// TIA Portal V17 export
// export: Created 2024-09-27T18:53:45.8218264Z, ExportSetting WithDefaults, DisplayName Totally Integrated Automation Portal, DisplayVersion V17, DisplayName TIA Portal Openness, DisplayVersion V17, DisplayName TIA Portal Version Control Interface, DisplayVersion V17, DisplayName STEP 7 Professional, DisplayVersion V17, DisplayName STEP 7 Safety, DisplayVersion V17, DisplayName WinCC Professional, DisplayVersion V17
FUNCTION "USTAWIENIA" : Void   // FC3, LAD
{ S7_Optimized_Access := 'TRUE' }
VERSION : 0.1
// stored: AutoNumber true, IsIECCheckEnabled false, SetENOAutomatically false, UDAEnableTagReadback false
   VAR_TEMP
      temp_calc_new_tact2 : DInt;
      temp_calc_3 : DInt;
      temp_calc4 : Real;
      temp_calc5 : DInt;
      temp_calc6 : DInt;
      m_zboczeP_ustaw_czas_ssania : Bool;
      temp_calc7 : Real;
      temp_calc8 : Real;
      temp_calc9 : Real;
      temp_calc10 : DInt;
      temp_calc11 : DInt;
      temp_calc12 : Real;
      temp_calc13 : Real;
      temp_calc14 : DInt;
      temp_calc15 : DInt;
      temp_calc16 : Real;
      temp_calc17 : Real;
      temp_calc18 : DInt;
      temp_calc19 : DInt;
      temp_calc20 : Real;
      m_zboczeN_ustaw_delay_zag : Bool;
      m_zboczeN_ustaw_delay_odb : Bool;
      m_zbocze_P_ustaw_delay_odbior : Bool;
   END_VAR
   VAR_TEMP   // added for the SCL form of the ladder/FBD networks
      _w1 : Bool;
      _w2 : Bool;
      _w3 : Bool;
      _w4 : Bool;
      _w5 : Bool;
      _w6 : Bool;
   END_VAR
BEGIN

REGION Network 1: KASOWANIE LICZNIKÓW ZADANYCH SZTUK I WYKONANYCH
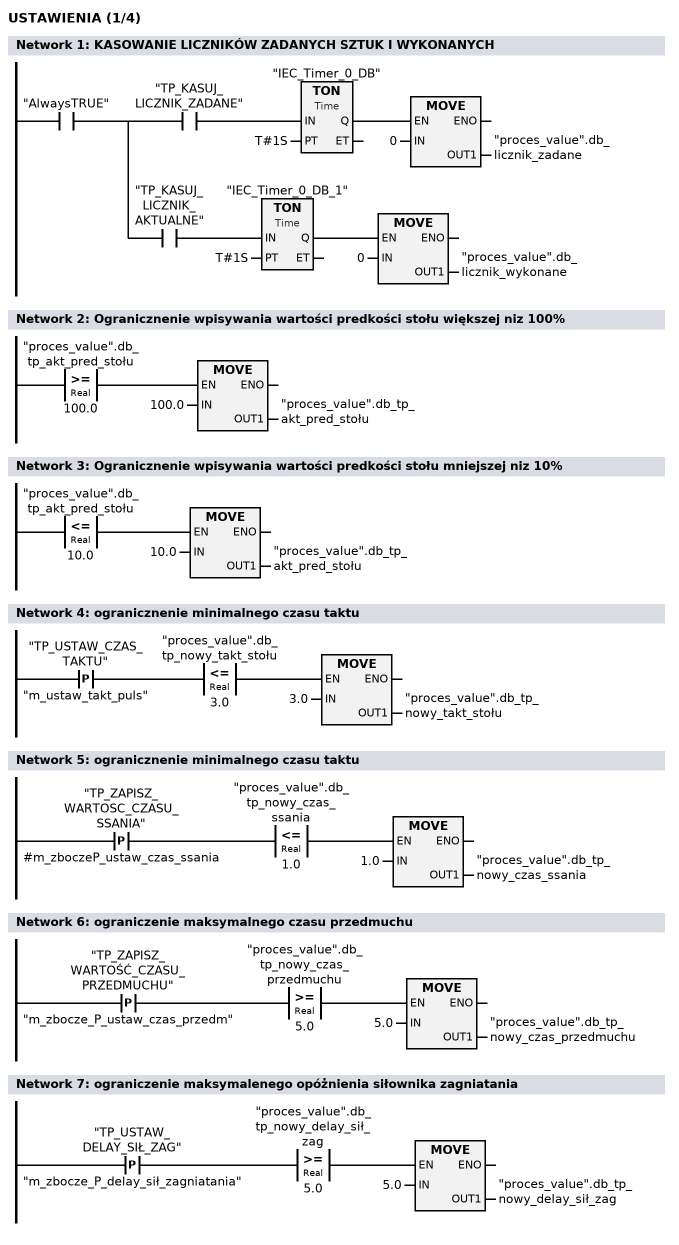
   RUNG wire#powerrail
      Contact( "AlwaysTRUE" )
      wire#w1
      Contact( "TP_KASUJ_LICZNIK_ZADANE" )
      { S7_Templates := "time_type := Time" } "IEC_Timer_0_DB".TON(pt := T#1S, et =>)
      Move(in := 0, out1 => "proces_value".db_licznik_zadane)
   END_RUNG
   RUNG wire#w1
      Contact( "TP_KASUJ_LICZNIK_AKTUALNE" )
      { S7_Templates := "time_type := Time" } "IEC_Timer_0_DB_1".TON(pt := T#1S, et =>)
      Move(in := 0, out1 => "proces_value".db_licznik_wykonane)
   END_RUNG
   // the same network as SCL:
   "IEC_Timer_0_DB".TON(IN := "AlwaysTRUE" AND "TP_KASUJ_LICZNIK_ZADANE", PT := T#1S);
   IF "IEC_Timer_0_DB".Q THEN "proces_value".db_licznik_zadane := 0; END_IF;
   "IEC_Timer_0_DB_1".TON(IN := "AlwaysTRUE" AND "TP_KASUJ_LICZNIK_AKTUALNE", PT := T#1S);
   IF "IEC_Timer_0_DB_1".Q THEN "proces_value".db_licznik_wykonane := 0; END_IF;
END_REGION

REGION Network 2: Ogranicznenie wpisywania wartości predkości stołu większej niz 100%
   RUNG wire#powerrail
      { S7_Templates := "SrcType := Real" } GE_Contact(in1 := "proces_value".db_tp_akt_pred_stołu, in2 := 100.0)
      Move(in := 100.0, out1 => "proces_value".db_tp_akt_pred_stołu)
   END_RUNG
   // the same network as SCL:
   IF "proces_value".db_tp_akt_pred_stołu >= 100.0 THEN "proces_value".db_tp_akt_pred_stołu := 100.0; END_IF;
END_REGION

REGION Network 3: Ogranicznenie wpisywania wartości predkości stołu mniejszej niz 10%
   RUNG wire#powerrail
      { S7_Templates := "SrcType := Real" } LE_Contact(in1 := "proces_value".db_tp_akt_pred_stołu, in2 := 10.0)
      Move(in := 10.0, out1 => "proces_value".db_tp_akt_pred_stołu)
   END_RUNG
   // the same network as SCL:
   IF "proces_value".db_tp_akt_pred_stołu <= 10.0 THEN "proces_value".db_tp_akt_pred_stołu := 10.0; END_IF;
END_REGION

REGION Network 4: ogranicznenie minimalnego czasu taktu
   RUNG wire#powerrail
      P_Contact(operand := "TP_USTAW_CZAS_TAKTU", bit := "m_ustaw_takt_puls")
      { S7_Templates := "SrcType := Real" } LE_Contact(in1 := "proces_value".db_tp_nowy_takt_stołu, in2 := 3.0)
      Move(in := 3.0, out1 => "proces_value".db_tp_nowy_takt_stołu)
   END_RUNG
   // the same network as SCL:
   #_w1 := "TP_USTAW_CZAS_TAKTU" AND NOT "m_ustaw_takt_puls";   // rising edge of "TP_USTAW_CZAS_TAKTU"
   "m_ustaw_takt_puls" := "TP_USTAW_CZAS_TAKTU";
   IF #_w1 AND ("proces_value".db_tp_nowy_takt_stołu <= 3.0) THEN
       "proces_value".db_tp_nowy_takt_stołu := 3.0;
   END_IF;
END_REGION

REGION Network 5: ogranicznenie minimalnego czasu taktu
   RUNG wire#powerrail
      P_Contact(operand := "TP_ZAPISZ_WARTOSC_CZASU_SSANIA", bit := #m_zboczeP_ustaw_czas_ssania)
      { S7_Templates := "SrcType := Real" } LE_Contact(in1 := "proces_value".db_tp_nowy_czas_ssania, in2 := 1.0)
      Move(in := 1.0, out1 => "proces_value".db_tp_nowy_czas_ssania)
   END_RUNG
   // the same network as SCL:
   #_w1 := "TP_ZAPISZ_WARTOSC_CZASU_SSANIA" AND NOT #m_zboczeP_ustaw_czas_ssania;   // rising edge of "TP_ZAPISZ_WARTOSC_CZASU_SSANIA"
   #m_zboczeP_ustaw_czas_ssania := "TP_ZAPISZ_WARTOSC_CZASU_SSANIA";
   IF #_w1 AND ("proces_value".db_tp_nowy_czas_ssania <= 1.0) THEN
       "proces_value".db_tp_nowy_czas_ssania := 1.0;
   END_IF;
END_REGION

REGION Network 6: ograniczenie maksymalnego czasu przedmuchu
   RUNG wire#powerrail
      P_Contact(operand := "TP_ZAPISZ_WARTOŚĆ_CZASU_PRZEDMUCHU", bit := "m_zbocze_P_ustaw_czas_przedm")
      { S7_Templates := "SrcType := Real" } GE_Contact(in1 := "proces_value".db_tp_nowy_czas_przedmuchu, in2 := 5.0)
      Move(in := 5.0, out1 => "proces_value".db_tp_nowy_czas_przedmuchu)
   END_RUNG
   // the same network as SCL:
   #_w1 := "TP_ZAPISZ_WARTOŚĆ_CZASU_PRZEDMUCHU" AND NOT "m_zbocze_P_ustaw_czas_przedm";   // rising edge of "TP_ZAPISZ_WARTOŚĆ_CZASU_PRZEDMUCHU"
   "m_zbocze_P_ustaw_czas_przedm" := "TP_ZAPISZ_WARTOŚĆ_CZASU_PRZEDMUCHU";
   IF #_w1 AND ("proces_value".db_tp_nowy_czas_przedmuchu >= 5.0) THEN
       "proces_value".db_tp_nowy_czas_przedmuchu := 5.0;
   END_IF;
END_REGION

REGION Network 7: ograniczenie maksymalenego opóżnienia siłownika zagniatania
   RUNG wire#powerrail
      P_Contact(operand := "TP_USTAW_DELAY_SIŁ_ZAG", bit := "m_zbocze_P_delay_sił_zagniatania")
      { S7_Templates := "SrcType := Real" } GE_Contact(in1 := "proces_value".db_tp_nowy_delay_sił_zag, in2 := 5.0)
      Move(in := 5.0, out1 => "proces_value".db_tp_nowy_delay_sił_zag)
   END_RUNG
   // the same network as SCL:
   #_w1 := "TP_USTAW_DELAY_SIŁ_ZAG" AND NOT "m_zbocze_P_delay_sił_zagniatania";   // rising edge of "TP_USTAW_DELAY_SIŁ_ZAG"
   "m_zbocze_P_delay_sił_zagniatania" := "TP_USTAW_DELAY_SIŁ_ZAG";
   IF #_w1 AND ("proces_value".db_tp_nowy_delay_sił_zag >= 5.0) THEN
       "proces_value".db_tp_nowy_delay_sił_zag := 5.0;
   END_IF;
END_REGION

REGION Network 8: ograniczenie maksymalenego opóżnienia siłownika odbioru
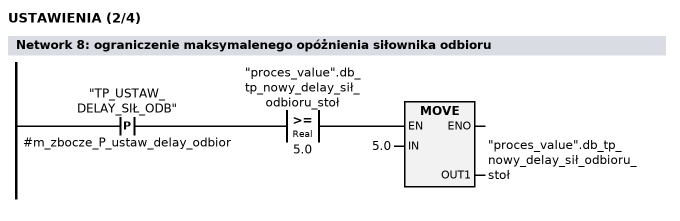
   RUNG wire#powerrail
      P_Contact(operand := "TP_USTAW_DELAY_SIŁ_ODB", bit := #m_zbocze_P_ustaw_delay_odbior)
      { S7_Templates := "SrcType := Real" } GE_Contact(in1 := "proces_value".db_tp_nowy_delay_sił_odbioru_stoł, in2 := 5.0)
      Move(in := 5.0, out1 => "proces_value".db_tp_nowy_delay_sił_odbioru_stoł)
   END_RUNG
   // the same network as SCL:
   #_w1 := "TP_USTAW_DELAY_SIŁ_ODB" AND NOT #m_zbocze_P_ustaw_delay_odbior;   // rising edge of "TP_USTAW_DELAY_SIŁ_ODB"
   #m_zbocze_P_ustaw_delay_odbior := "TP_USTAW_DELAY_SIŁ_ODB";
   IF #_w1 AND ("proces_value".db_tp_nowy_delay_sił_odbioru_stoł >= 5.0) THEN
       "proces_value".db_tp_nowy_delay_sił_odbioru_stoł := 5.0;
   END_IF;
END_REGION

REGION Network 9: OBSŁUGA LICZNIKÓW I TIMERÓW
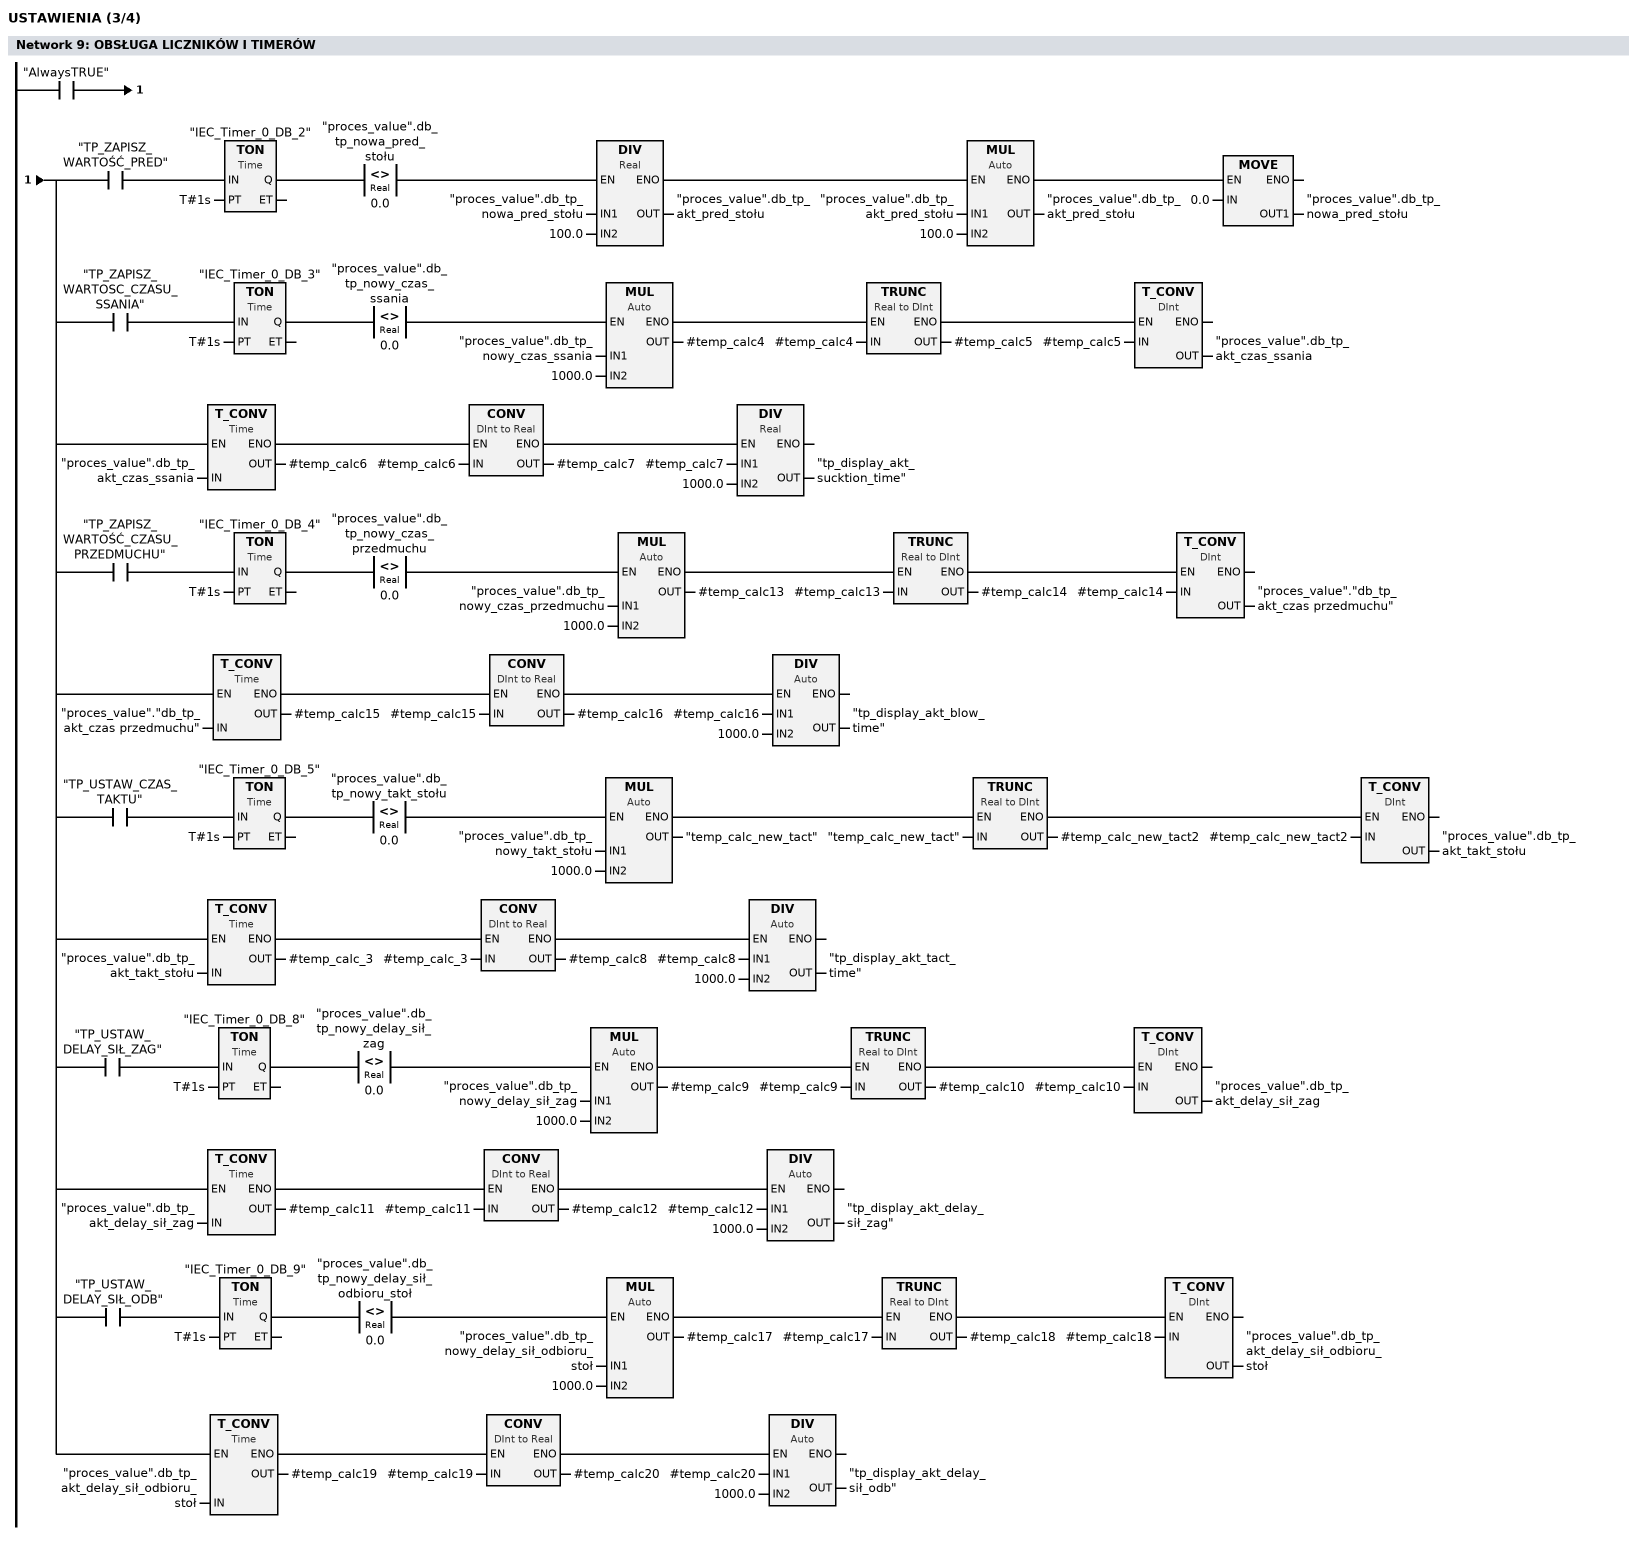
   RUNG wire#powerrail
      Contact( "AlwaysTRUE" )
      wire#w1
      Contact( "TP_ZAPISZ_WARTOŚĆ_PRED" )
      { S7_Templates := "time_type := Time" } "IEC_Timer_0_DB_2".TON(pt := T#1s, et =>)
      { S7_Templates := "SrcType := Real" } NE_Contact(in1 := "proces_value".db_tp_nowa_pred_stołu, in2 := 0.0)
      { S7_Templates := "SrcType := Real" } Div(in1 := "proces_value".db_tp_nowa_pred_stołu, in2 := 100.0, out => "proces_value".db_tp_akt_pred_stołu)
      Mul(in1 := "proces_value".db_tp_akt_pred_stołu, in2 := 100.0, out => "proces_value".db_tp_akt_pred_stołu)
      Move(in := 0.0, out1 => "proces_value".db_tp_nowa_pred_stołu)
   END_RUNG
   RUNG wire#w1
      Contact( "TP_ZAPISZ_WARTOSC_CZASU_SSANIA" )
      { S7_Templates := "time_type := Time" } "IEC_Timer_0_DB_3".TON(pt := T#1s, et =>)
      { S7_Templates := "SrcType := Real" } NE_Contact(in1 := "proces_value".db_tp_nowy_czas_ssania, in2 := 0.0)
      Mul(in1 := "proces_value".db_tp_nowy_czas_ssania, in2 := 1000.0, out => #temp_calc4)
      { S7_Templates := "[SrcType := Real, DestType := DInt]" } Trunc(in := #temp_calc4, out => #temp_calc5)
      { S7_Templates := "[src_type := DInt, dest_type := Time]" } T_CONV(IN := #temp_calc5, OUT => "proces_value".db_tp_akt_czas_ssania)
   END_RUNG
   RUNG wire#w1
      { S7_Templates := "[src_type := Time, dest_type := DInt]" } T_CONV(IN := "proces_value".db_tp_akt_czas_ssania, OUT => #temp_calc6)
      { S7_Templates := "[SrcType := DInt, DestType := Real]" } Convert(in := #temp_calc6, out => #temp_calc7)
      { S7_Templates := "SrcType := Real" } Div(in1 := #temp_calc7, in2 := 1000.0, out => "tp_display_akt_sucktion_time")
   END_RUNG
   RUNG wire#w1
      Contact( "TP_ZAPISZ_WARTOŚĆ_CZASU_PRZEDMUCHU" )
      { S7_Templates := "time_type := Time" } "IEC_Timer_0_DB_4".TON(pt := T#1s, et =>)
      { S7_Templates := "SrcType := Real" } NE_Contact(in1 := "proces_value".db_tp_nowy_czas_przedmuchu, in2 := 0.0)
      Mul(in1 := "proces_value".db_tp_nowy_czas_przedmuchu, in2 := 1000.0, out => #temp_calc13)
      { S7_Templates := "[SrcType := Real, DestType := DInt]" } Trunc(in := #temp_calc13, out => #temp_calc14)
      { S7_Templates := "[src_type := DInt, dest_type := Time]" } T_CONV(IN := #temp_calc14, OUT => "proces_value"."db_tp_akt_czas przedmuchu")
   END_RUNG
   RUNG wire#w1
      { S7_Templates := "[src_type := Time, dest_type := DInt]" } T_CONV(IN := "proces_value"."db_tp_akt_czas przedmuchu", OUT => #temp_calc15)
      { S7_Templates := "[SrcType := DInt, DestType := Real]" } Convert(in := #temp_calc15, out => #temp_calc16)
      Div(in1 := #temp_calc16, in2 := 1000.0, out => "tp_display_akt_blow_time")
   END_RUNG
   RUNG wire#w1
      Contact( "TP_USTAW_CZAS_TAKTU" )
      { S7_Templates := "time_type := Time" } "IEC_Timer_0_DB_5".TON(pt := T#1s, et =>)
      { S7_Templates := "SrcType := Real" } NE_Contact(in1 := "proces_value".db_tp_nowy_takt_stołu, in2 := 0.0)
      Mul(in1 := "proces_value".db_tp_nowy_takt_stołu, in2 := 1000.0, out => "temp_calc_new_tact")
      { S7_Templates := "[SrcType := Real, DestType := DInt]" } Trunc(in := "temp_calc_new_tact", out => #temp_calc_new_tact2)
      { S7_Templates := "[src_type := DInt, dest_type := Time]" } T_CONV(IN := #temp_calc_new_tact2, OUT => "proces_value".db_tp_akt_takt_stołu)
   END_RUNG
   RUNG wire#w1
      { S7_Templates := "[src_type := Time, dest_type := DInt]" } T_CONV(IN := "proces_value".db_tp_akt_takt_stołu, OUT => #temp_calc_3)
      { S7_Templates := "[SrcType := DInt, DestType := Real]" } Convert(in := #temp_calc_3, out => #temp_calc8)
      Div(in1 := #temp_calc8, in2 := 1000.0, out => "tp_display_akt_tact_time")
   END_RUNG
   RUNG wire#w1
      Contact( "TP_USTAW_DELAY_SIŁ_ZAG" )
      { S7_Templates := "time_type := Time" } "IEC_Timer_0_DB_8".TON(pt := T#1s, et =>)
      { S7_Templates := "SrcType := Real" } NE_Contact(in1 := "proces_value".db_tp_nowy_delay_sił_zag, in2 := 0.0)
      Mul(in1 := "proces_value".db_tp_nowy_delay_sił_zag, in2 := 1000.0, out => #temp_calc9)
      { S7_Templates := "[SrcType := Real, DestType := DInt]" } Trunc(in := #temp_calc9, out => #temp_calc10)
      { S7_Templates := "[src_type := DInt, dest_type := Time]" } T_CONV(IN := #temp_calc10, OUT => "proces_value".db_tp_akt_delay_sił_zag)
   END_RUNG
   RUNG wire#w1
      { S7_Templates := "[src_type := Time, dest_type := DInt]" } T_CONV(IN := "proces_value".db_tp_akt_delay_sił_zag, OUT => #temp_calc11)
      { S7_Templates := "[SrcType := DInt, DestType := Real]" } Convert(in := #temp_calc11, out => #temp_calc12)
      Div(in1 := #temp_calc12, in2 := 1000.0, out => "tp_display_akt_delay_sił_zag")
   END_RUNG
   RUNG wire#w1
      Contact( "TP_USTAW_DELAY_SIŁ_ODB" )
      { S7_Templates := "time_type := Time" } "IEC_Timer_0_DB_9".TON(pt := T#1s, et =>)
      { S7_Templates := "SrcType := Real" } NE_Contact(in1 := "proces_value".db_tp_nowy_delay_sił_odbioru_stoł, in2 := 0.0)
      Mul(in1 := "proces_value".db_tp_nowy_delay_sił_odbioru_stoł, in2 := 1000.0, out => #temp_calc17)
      { S7_Templates := "[SrcType := Real, DestType := DInt]" } Trunc(in := #temp_calc17, out => #temp_calc18)
      { S7_Templates := "[src_type := DInt, dest_type := Time]" } T_CONV(IN := #temp_calc18, OUT => "proces_value".db_tp_akt_delay_sił_odbioru_stoł)
   END_RUNG
   RUNG wire#w1
      { S7_Templates := "[src_type := Time, dest_type := DInt]" } T_CONV(IN := "proces_value".db_tp_akt_delay_sił_odbioru_stoł, OUT => #temp_calc19)
      { S7_Templates := "[SrcType := DInt, DestType := Real]" } Convert(in := #temp_calc19, out => #temp_calc20)
      Div(in1 := #temp_calc20, in2 := 1000.0, out => "tp_display_akt_delay_sił_odb")
   END_RUNG
   // the same network as SCL:
   "IEC_Timer_0_DB_2".TON(IN := "AlwaysTRUE" AND "TP_ZAPISZ_WARTOŚĆ_PRED", PT := T#1s);
   IF "IEC_Timer_0_DB_2".Q AND ("proces_value".db_tp_nowa_pred_stołu <> 0.0) THEN
       "proces_value".db_tp_akt_pred_stołu := "proces_value".db_tp_nowa_pred_stołu / 100.0;
       "proces_value".db_tp_akt_pred_stołu := "proces_value".db_tp_akt_pred_stołu * 100.0;
       "proces_value".db_tp_nowa_pred_stołu := 0.0;
   END_IF;
   "IEC_Timer_0_DB_3".TON(IN := "AlwaysTRUE" AND "TP_ZAPISZ_WARTOSC_CZASU_SSANIA", PT := T#1s);
   IF "IEC_Timer_0_DB_3".Q AND ("proces_value".db_tp_nowy_czas_ssania <> 0.0) THEN
       #temp_calc4 := "proces_value".db_tp_nowy_czas_ssania * 1000.0;
       #temp_calc5 := TRUNC(#temp_calc4);
   END_IF;
   #_w1 := "AlwaysTRUE";
   IF "IEC_Timer_0_DB_3".Q AND ("proces_value".db_tp_nowy_czas_ssania <> 0.0) THEN
       T_CONV(IN := #temp_calc5, OUT => "proces_value".db_tp_akt_czas_ssania);
   END_IF;
   T_CONV(EN := #_w1, IN := "proces_value".db_tp_akt_czas_ssania, OUT => #temp_calc6, ENO => #_w2);
   IF #_w2 THEN
       #temp_calc7 := DINT_TO_REAL(#temp_calc6);
       "tp_display_akt_sucktion_time" := #temp_calc7 / 1000.0;
   END_IF;
   "IEC_Timer_0_DB_4".TON(IN := #_w1 AND "TP_ZAPISZ_WARTOŚĆ_CZASU_PRZEDMUCHU", PT := T#1s);
   IF "IEC_Timer_0_DB_4".Q AND ("proces_value".db_tp_nowy_czas_przedmuchu <> 0.0) THEN
       #temp_calc13 := "proces_value".db_tp_nowy_czas_przedmuchu * 1000.0;
       #temp_calc14 := TRUNC(#temp_calc13);
       T_CONV(IN := #temp_calc14, OUT => "proces_value"."db_tp_akt_czas przedmuchu");
   END_IF;
   T_CONV(EN := #_w1, IN := "proces_value"."db_tp_akt_czas przedmuchu", OUT => #temp_calc15, ENO => #_w3);
   IF #_w3 THEN
       #temp_calc16 := DINT_TO_REAL(#temp_calc15);
       "tp_display_akt_blow_time" := #temp_calc16 / 1000.0;
   END_IF;
   "IEC_Timer_0_DB_5".TON(IN := #_w1 AND "TP_USTAW_CZAS_TAKTU", PT := T#1s);
   IF "IEC_Timer_0_DB_5".Q AND ("proces_value".db_tp_nowy_takt_stołu <> 0.0) THEN
       "temp_calc_new_tact" := "proces_value".db_tp_nowy_takt_stołu * 1000.0;
       #temp_calc_new_tact2 := TRUNC("temp_calc_new_tact");
       T_CONV(IN := #temp_calc_new_tact2, OUT => "proces_value".db_tp_akt_takt_stołu);
   END_IF;
   T_CONV(EN := #_w1, IN := "proces_value".db_tp_akt_takt_stołu, OUT => #temp_calc_3, ENO => #_w4);
   IF #_w4 THEN
       #temp_calc8 := DINT_TO_REAL(#temp_calc_3);
       "tp_display_akt_tact_time" := #temp_calc8 / 1000.0;
   END_IF;
   "IEC_Timer_0_DB_8".TON(IN := #_w1 AND "TP_USTAW_DELAY_SIŁ_ZAG", PT := T#1s);
   IF "IEC_Timer_0_DB_8".Q AND ("proces_value".db_tp_nowy_delay_sił_zag <> 0.0) THEN
       #temp_calc9 := "proces_value".db_tp_nowy_delay_sił_zag * 1000.0;
       #temp_calc10 := TRUNC(#temp_calc9);
       T_CONV(IN := #temp_calc10, OUT => "proces_value".db_tp_akt_delay_sił_zag);
   END_IF;
   T_CONV(EN := #_w1, IN := "proces_value".db_tp_akt_delay_sił_zag, OUT => #temp_calc11, ENO => #_w5);
   IF #_w5 THEN
       #temp_calc12 := DINT_TO_REAL(#temp_calc11);
       "tp_display_akt_delay_sił_zag" := #temp_calc12 / 1000.0;
   END_IF;
   "IEC_Timer_0_DB_9".TON(IN := #_w1 AND "TP_USTAW_DELAY_SIŁ_ODB", PT := T#1s);
   IF "IEC_Timer_0_DB_9".Q AND ("proces_value".db_tp_nowy_delay_sił_odbioru_stoł <> 0.0) THEN
       #temp_calc17 := "proces_value".db_tp_nowy_delay_sił_odbioru_stoł * 1000.0;
       #temp_calc18 := TRUNC(#temp_calc17);
       T_CONV(IN := #temp_calc18, OUT => "proces_value".db_tp_akt_delay_sił_odbioru_stoł);
   END_IF;
   T_CONV(EN := #_w1, IN := "proces_value".db_tp_akt_delay_sił_odbioru_stoł, OUT => #temp_calc19, ENO => #_w6);
   IF #_w6 THEN
       #temp_calc20 := DINT_TO_REAL(#temp_calc19);
       "tp_display_akt_delay_sił_odb" := #temp_calc20 / 1000.0;
   END_IF;
END_REGION

REGION Network 10: podswietlenie przycisku po ustawieniu gniazda płytkiego jako 1
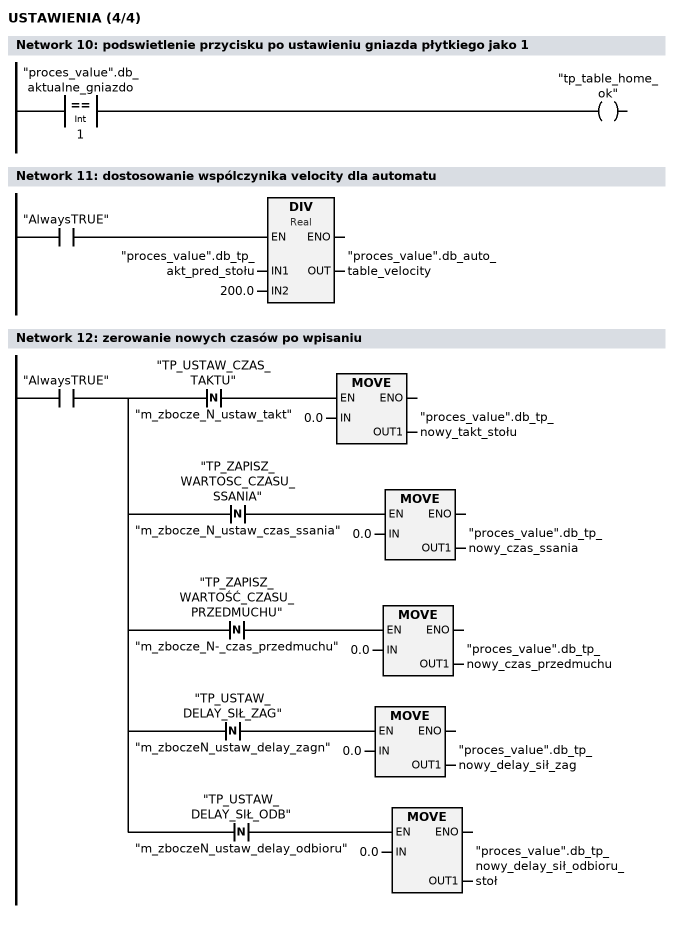
   RUNG wire#powerrail
      { S7_Templates := "SrcType := Int" } EQ_Contact(in1 := "proces_value".db_aktualne_gniazdo, in2 := 1)
      Coil( "tp_table_home_ok" )
   END_RUNG
   // the same network as SCL:
   "tp_table_home_ok" := "proces_value".db_aktualne_gniazdo = 1;
END_REGION

REGION Network 11: dostosowanie wspólczynika velocity dla automatu
   RUNG wire#powerrail
      Contact( "AlwaysTRUE" )
      { S7_Templates := "SrcType := Real" } Div(in1 := "proces_value".db_tp_akt_pred_stołu, in2 := 200.0, out => "proces_value".db_auto_table_velocity)
   END_RUNG
   // the same network as SCL:
   IF "AlwaysTRUE" THEN
       "proces_value".db_auto_table_velocity := "proces_value".db_tp_akt_pred_stołu / 200.0;
   END_IF;
END_REGION

REGION Network 12: zerowanie nowych czasów po wpisaniu
   RUNG wire#powerrail
      Contact( "AlwaysTRUE" )
      wire#w1
      N_Contact(operand := "TP_USTAW_CZAS_TAKTU", bit := "m_zbocze_N_ustaw_takt")
      Move(in := 0.0, out1 => "proces_value".db_tp_nowy_takt_stołu)
   END_RUNG
   RUNG wire#w1
      N_Contact(operand := "TP_ZAPISZ_WARTOSC_CZASU_SSANIA", bit := "m_zbocze_N_ustaw_czas_ssania")
      Move(in := 0.0, out1 => "proces_value".db_tp_nowy_czas_ssania)
   END_RUNG
   RUNG wire#w1
      N_Contact(operand := "TP_ZAPISZ_WARTOŚĆ_CZASU_PRZEDMUCHU", bit := "m_zbocze_N-_czas_przedmuchu")
      Move(in := 0.0, out1 => "proces_value".db_tp_nowy_czas_przedmuchu)
   END_RUNG
   RUNG wire#w1
      N_Contact(operand := "TP_USTAW_DELAY_SIŁ_ZAG", bit := "m_zboczeN_ustaw_delay_zagn")
      Move(in := 0.0, out1 => "proces_value".db_tp_nowy_delay_sił_zag)
   END_RUNG
   RUNG wire#w1
      N_Contact(operand := "TP_USTAW_DELAY_SIŁ_ODB", bit := "m_zboczeN_ustaw_delay_odbioru")
      Move(in := 0.0, out1 => "proces_value".db_tp_nowy_delay_sił_odbioru_stoł)
   END_RUNG
   // the same network as SCL:
   #_w1 := "AlwaysTRUE" AND NOT "TP_USTAW_CZAS_TAKTU" AND "m_zbocze_N_ustaw_takt";   // falling edge of "TP_USTAW_CZAS_TAKTU"
   "m_zbocze_N_ustaw_takt" := "TP_USTAW_CZAS_TAKTU";
   IF #_w1 THEN "proces_value".db_tp_nowy_takt_stołu := 0.0; END_IF;
   #_w2 := "AlwaysTRUE" AND NOT "TP_ZAPISZ_WARTOSC_CZASU_SSANIA" AND "m_zbocze_N_ustaw_czas_ssania";   // falling edge of "TP_ZAPISZ_WARTOSC_CZASU_SSANIA"
   "m_zbocze_N_ustaw_czas_ssania" := "TP_ZAPISZ_WARTOSC_CZASU_SSANIA";
   IF #_w2 THEN "proces_value".db_tp_nowy_czas_ssania := 0.0; END_IF;
   #_w3 := "AlwaysTRUE" AND NOT "TP_ZAPISZ_WARTOŚĆ_CZASU_PRZEDMUCHU" AND "m_zbocze_N-_czas_przedmuchu";   // falling edge of "TP_ZAPISZ_WARTOŚĆ_CZASU_PRZEDMUCHU"
   "m_zbocze_N-_czas_przedmuchu" := "TP_ZAPISZ_WARTOŚĆ_CZASU_PRZEDMUCHU";
   IF #_w3 THEN "proces_value".db_tp_nowy_czas_przedmuchu := 0.0; END_IF;
   #_w4 := "AlwaysTRUE" AND NOT "TP_USTAW_DELAY_SIŁ_ZAG" AND "m_zboczeN_ustaw_delay_zagn";   // falling edge of "TP_USTAW_DELAY_SIŁ_ZAG"
   "m_zboczeN_ustaw_delay_zagn" := "TP_USTAW_DELAY_SIŁ_ZAG";
   IF #_w4 THEN "proces_value".db_tp_nowy_delay_sił_zag := 0.0; END_IF;
   #_w5 := "AlwaysTRUE" AND NOT "TP_USTAW_DELAY_SIŁ_ODB" AND "m_zboczeN_ustaw_delay_odbioru";   // falling edge of "TP_USTAW_DELAY_SIŁ_ODB"
   "m_zboczeN_ustaw_delay_odbioru" := "TP_USTAW_DELAY_SIŁ_ODB";
   IF #_w5 THEN "proces_value".db_tp_nowy_delay_sił_odbioru_stoł := 0.0; END_IF;
END_REGION
END_FUNCTION
